PROGRAM MAIN
VAR
    sdValve : SD_Valve;
    openCmd : BOOL;
    openResult : BOOL;
    closeCmd : BOOL;
    closeResult : BOOL;
    goToAutoCmd : BOOL;
    goToManaulCmd : BOOL;
    goToInitCmd : BOOL;
END_VAR

sdValve();

IF openCmd THEN
    openCmd := FALSE;
    openResult := FALSE;
    openResult :=sdValve.OpenValve();
END_IF

IF closeCmd THEN
    closeCmd := FALSE;
    closeResult := FALSE;
    closeResult := sdValve.CloseValve();
END_IF

IF goToAutoCmd THEN
    goToAutoCmd := FALSE;
    sdValve.GoToAutoState();
END_IF

IF goToManaulCmd THEN
    goToManaulCmd := FALSE;
    sdValve.GoToManualState();
END_IF

IF goToInitCmd THEN
    goToInitCmd := FALSE;
    sdValve.GoToInitState();
END_IF

END_PROGRAM

(* stored: Version 1.1.0.1, ProductVersion 3.1.4024.12
   POU MAIN: Id {8dd93341-7f75-4066-b92e-0123e424ddd6}, SpecialFunc None *)
